(* CODESYS project OpenSML_TC3.library
   Company: Github
   DefaultNamespace: OpenSML
   Version: 3.2
   Placeholder: OpenSML
   Author: Feecat
   Description: Open Sources SoftMotion Light For CiA402 Servo Drivers
      visit https://github.com/feecat/OpenSML for more information
   Title: OpenSML

Project tree, tasks and I/O mapping:
  libraries: Tc2_Standard, * (Beckhoff Automation GmbH)
  S7RTT/
    function block FB_S7RTT_OTG [ST]
    function block FB_S7RTT_Plan [ST]
    function FC_S7RTT_AtTime [ST]
    function FC_S7RTT_BuildProfile [ST]
    function FC_S7RTT_CalcTrajDist [ST]
    data type ST_MotionLimits
    data type ST_MotionState
  data type OpenSML_Axis
  function block OpenSML_AxisController [ST]
  data type OpenSML_Control
  function block OpenSML_Home [ST]
  function block OpenSML_Power [ST]
  function block OpenSML_ProfilePosition [ST]
  function block OpenSML_ProfileVelocity [ST]
  function block OpenSML_Stop [ST]
  function block OpenSML_SyncPosition [ST]
  function block OpenSML_SyncVelocity [ST]
  function block OpenSML_TC3Link [ST]
*)

// S7RTT/ST_MotionLimits
TYPE ST_MotionLimits :
STRUCT
	fVelMax: LREAL;
	fAccMax: LREAL;
	fJerkMax: LREAL;
END_STRUCT
END_TYPE

// S7RTT/ST_MotionState
TYPE ST_MotionState :
STRUCT
	/// Duration of this segment 
	fDuration: LREAL := 0.0;
	/// Position 
	fPos: LREAL := 0.0;
	/// Velocity 
	fVel: LREAL := 0.0;
	/// Acceleration 
	fAcc: LREAL := 0.0;
	/// Jerk 
	fJerk: LREAL := 0.0;
END_STRUCT
END_TYPE

// OpenSML_Axis
TYPE OpenSML_Axis :
STRUCT
	///Output
	ControlWord: UINT;
	Modes_of_operation: SINT;
	Target_Position: DINT;
	Profile_Velocity: UDINT;
	Target_Velocity: DINT;
	Target_torque: INT;
	///Input
	StatusWord: UINT;
	Modes_of_operation_display: SINT;
	Torque_Actual_Value: INT;
	Position_Actual_Value: DINT;
	Velocity_Actual_Value: DINT;
	Current_Actual_Value: INT;
	Following_Error_Actual_Value: DINT;
END_STRUCT
END_TYPE

// OpenSML_Control
TYPE OpenSML_Control :
STRUCT
	///Axis Hardware Enable
	xAxisEnable: BOOL;
	///Jog&Pos Movement Enable
	xMoveEnable: BOOL;
	///Home Function Enable
	xHomeEnable: BOOL;
	///Simulation Mode
	xSimulation: BOOL;
	///Emergency Stop
	xEmergencyStop: BOOL := TRUE;
	///Jog Positive
	JogPos: BOOL;
	///Jog Negative
	JogNeg: BOOL;
	///Jog Velocity
	JogVelocity: LREAL := 10;
	///Actual Position Feedback
	lrActualPosition: LREAL;
	///Follow Target Position, Can be set to new value at any time
	lrFollowPosition: LREAL;
	///Follow Move Velocity, Can be set to new value at any time
	lrFollowVelocity: LREAL := 20;
	///Follow Move Enable
	xFollowEnable: BOOL;
	///Error
	xError: BOOL;
	///Busy, Normal Working State
	xBusy: BOOL;
	///In Position
	xInPosition: BOOL;
	///Axis Hardware Enabled
	xEnabled: BOOL;
	///Axis Home Done
	xHomeDone: BOOL;
	///Max Velocity
	MaxVelocity: LREAL := 100;
	///Max Acceleration
	MaxAcceleration: LREAL := 1000;
	///Max Jerk
	MaxJerk: LREAL := 10000;
	///Task Cycle Time, 0.001 = 1ms
	CycleTime: LREAL := 0.001;
	///Scale
	Scale: LREAL := 16#1000;
	///Axis Reference
	Axis: OpenSML_Axis;
END_STRUCT
END_TYPE

// S7RTT/FB_S7RTT_OTG
FUNCTION_BLOCK FB_S7RTT_OTG
VAR_INPUT
	///false=position, true=velocity
	ControlInterface: BOOL := FALSE;
	TargetPosition: LREAL;
	TargetVelocity: LREAL := 0;
	///1ms
	CycleTime: LREAL := 0.001;
	MaxVelocity: LREAL := 10;
	MaxAcceleration: LREAL := 10;
	MaxJerk: LREAL := 10;
	///set when init
	CurrentPosition: LREAL;
END_VAR
VAR_OUTPUT
	NewPosition: LREAL;
	NewVelocity: LREAL;
	NewAcceleration: LREAL;
	xError: BOOL;
END_VAR
VAR
	_ControlInterface: BOOL;
	_TargetPosition: LREAL;
	_TargetVelocity: LREAL;
	_CycleTime: LREAL;
	_MaxVelocity: LREAL;
	_MaxAcceleration: LREAL;
	_MaxJerk: LREAL;
	_CurrentPosition: LREAL;
	xExecute: BOOL;
	fbS7Planner: FB_S7RTT_Plan;
	stS7Limits: ST_MotionLimits;
	stS7Start: ST_MotionState;
	stS7Result: ST_MotionState;
	fS7Timer: LREAL;
END_VAR

// check if input changed
IF (ControlInterface <> _ControlInterface) OR
	(TargetPosition <> _TargetPosition) OR
	(TargetVelocity <> _TargetVelocity) OR
	(CycleTime <> _CycleTime) OR
	(MaxVelocity <> _MaxVelocity) OR
	(MaxAcceleration <> _MaxAcceleration) OR
	(MaxJerk <> _MaxJerk) OR
	(CurrentPosition <> _CurrentPosition) THEN
	
	IF CurrentPosition <> _CurrentPosition THEN
		stS7Start.fPos := CurrentPosition;
		stS7Result.fPos := CurrentPosition;
		_CurrentPosition := CurrentPosition;
	END_IF
	_ControlInterface := ControlInterface;
	_TargetPosition := TargetPosition;
	_TargetVelocity := TargetVelocity;
	_CycleTime := CycleTime;
	_MaxVelocity := MaxVelocity;
	_MaxAcceleration := MaxAcceleration;
	_MaxJerk := MaxJerk;
	
	xExecute:=TRUE;
END_IF

// main logic
IF xExecute THEN
    stS7Start.fPos := stS7Result.fPos;
    stS7Start.fVel := stS7Result.fVel;
    stS7Start.fAcc := stS7Result.fAcc;
    stS7Start.fDuration := 0.0;
    
    stS7Limits.fVelMax := MaxVelocity;
    stS7Limits.fAccMax := MaxAcceleration;
    stS7Limits.fJerkMax := MaxJerk;
    
    fbS7Planner.ModeVelocity := ControlInterface;
    fbS7Planner.StartState := stS7Start;
    fbS7Planner.TargetPos := TargetPosition;
    fbS7Planner.TargetVel := TargetVelocity; 
    fbS7Planner.Limits := stS7Limits;
    
    fS7Timer := 0.0;
END_IF

IF xExecute THEN
    fbS7Planner(Execute:=TRUE, Error=>xError);
    fbS7Planner(Execute:=FALSE);
END_IF

xExecute := FALSE;

fS7Timer := fS7Timer + CycleTime;

stS7Result := FC_S7RTT_AtTime(
	Trajectory := fbS7Planner.Trajectory, 
	SegCount := fbS7Planner.SegmentCount, 
	ElapsedTime := fS7Timer
);

NewPosition:=stS7Result.fPos;
NewVelocity:=stS7Result.fVel;
NewAcceleration:=stS7Result.fAcc;

END_FUNCTION_BLOCK

// S7RTT/FC_S7RTT_AtTime
FUNCTION FC_S7RTT_AtTime : ST_MotionState
VAR_INPUT
	Trajectory: ARRAY[1..32] OF ST_MotionState;
	SegCount: INT;
	ElapsedTime: LREAL;
END_VAR
VAR
	i: INT;
	t_rem: LREAL;
	t: LREAL;
	j: LREAL;
	p0: LREAL;
	v0: LREAL;
	a0: LREAL;
	last_idx: INT;
END_VAR

IF SegCount <= 0 THEN
    // No trajectory, return first state
    FC_S7RTT_AtTime.fPos := Trajectory[1].fPos; FC_S7RTT_AtTime.fVel := 0.0; FC_S7RTT_AtTime.fAcc := 0.0;
    RETURN;
END_IF;

IF ElapsedTime <= 0.0 THEN
     // Return Initial State from First Segment
     FC_S7RTT_AtTime := Trajectory[1]; 
     FC_S7RTT_AtTime.fDuration := 0.0;
     FC_S7RTT_AtTime.fJerk := 0.0;
     RETURN;
END_IF;

t_rem := ElapsedTime;

FOR i := 1 TO SegCount DO
	IF t_rem <= Trajectory[i].fDuration THEN
		t := t_rem;
		j := Trajectory[i].fJerk;
		// Use pre-calculated state at segment start
		p0 := Trajectory[i].fPos;
		v0 := Trajectory[i].fVel;
		a0 := Trajectory[i].fAcc;

		FC_S7RTT_AtTime.fPos := p0 + v0 * t + 0.5 * a0 * t*t + (1.0/6.0) * j * t*t*t;
		FC_S7RTT_AtTime.fVel := v0 + a0 * t + 0.5 * j * t*t;
		FC_S7RTT_AtTime.fAcc := a0 + j * t;
		FC_S7RTT_AtTime.fJerk := j;
		FC_S7RTT_AtTime.fDuration := 0.0;
		RETURN;
	ELSE
		t_rem := t_rem - Trajectory[i].fDuration;
	END_IF;
END_FOR;

// Time is beyond end of trajectory
// Calculate Final State of last segment
last_idx := SegCount;
t := Trajectory[last_idx].fDuration;
j := Trajectory[last_idx].fJerk;
p0 := Trajectory[last_idx].fPos;
v0 := Trajectory[last_idx].fVel;
a0 := Trajectory[last_idx].fAcc;

p0 := p0 + v0 * t + 0.5 * a0 * t*t + (1.0/6.0) * j * t*t*t;
v0 := v0 + a0 * t + 0.5 * j * t*t;

// Hold Final Position (assuming v=target, a=0 at end)
// Linear projection if Velocity is non-zero
FC_S7RTT_AtTime.fPos := p0 + v0 * t_rem;
FC_S7RTT_AtTime.fVel := v0;
FC_S7RTT_AtTime.fAcc := 0.0;
FC_S7RTT_AtTime.fJerk := 0.0;
FC_S7RTT_AtTime.fDuration := 0.0;

END_FUNCTION

// S7RTT/FB_S7RTT_Plan
FUNCTION_BLOCK FB_S7RTT_Plan
VAR_INPUT
	Execute: BOOL;
	ModeVelocity: BOOL;
	StartState: ST_MotionState;
	TargetPos: LREAL;
	TargetVel: LREAL;
	Limits: ST_MotionLimits;
END_VAR
VAR_OUTPUT
	Done: BOOL;
	Error: BOOL;
	SegmentCount: INT;
	Trajectory: ARRAY[1..32] OF ST_MotionState;
END_VAR
VAR
	/// State & Triggers
	trig_exec: BOOL;
	prev_exec: BOOL;
	c_pos: LREAL;
	c_vel: LREAL;
	c_acc: LREAL;
	/// Loop Iterators
	i: INT;
	/// Loop Iterators
	k: INT;
	/// General Calculation
	dist_req: LREAL;
	t_rec: LREAL;
	gap: LREAL;
	/// Check Bounds
	d_upper: LREAL;
	/// Check Bounds
	d_lower: LREAL;
	t_cruise: LREAL;
	/// --- Solver Shared Variables ---
	iter: INT;
	sa: LREAL;
	sb: LREAL;
	sc: LREAL;
	fa: LREAL;
	fb: LREAL;
	fc: LREAL;
	sd: LREAL;
	se: LREAL;
	tol1: LREAL;
	xm: LREAL;
	min1: LREAL;
	min2: LREAL;
	fCoefP: LREAL;
	fCoefQ: LREAL;
	fCoefR: LREAL;
	fCoefS: LREAL;
	mflag: BOOL;
	/// --- V1.7 Time Optimal Specific ---
	use_optimal: BOOL;
	opt_success: BOOL;
	/// 0 or 1
	j_idx: INT;
	j_apply: LREAL;
	search_horizon: LREAL;
	t_est: LREAL;
	/// Simulation / Cost Function Vars
	sim_p: LREAL;
	/// Simulation / Cost Function Vars
	sim_v: LREAL;
	/// Simulation / Cost Function Vars
	sim_a: LREAL;
	limit_a: LREAL;
	dist_to_lim: LREAL;
	t_ramp: LREAL;
	t_hold: LREAL;
	sat_dt: LREAL;
	sat_j: LREAL;
	/// Best Candidate Tracking
	valid_curr: BOOL;
	best_t_curr: LREAL;
	dur_curr: LREAL;
	winner_found: BOOL;
	winner_dur: LREAL;
	winner_t: LREAL;
	winner_j: LREAL;
	/// --- Fallback / Old Variables ---
	best_v: LREAL;
	v_mid: LREAL;
	a_mid: LREAL;
	v_inertial: LREAL;
	d_inertial: LREAL;
	t_to_zero: LREAL;
	j_restore: LREAL;
	/// Buffers
	t_shape_buf: ARRAY[1..5] OF LREAL;
	j_shape_buf: ARRAY[1..5] OF LREAL;
	shape_cnt: INT;
	/// Refinement
	ref_idx: INT;
	max_dt: LREAL;
	dt_fix: LREAL;
	v_cruise_start: LREAL;
	/// Constants (Updated V1.7)
	EPS_TIME: LREAL := 1E-10;
	/// Velocity Tolerance
	EPS_VAL: LREAL := 1E-10;
	EPS_ACC: LREAL := 1E-10;
	EPS_DIST: LREAL := 1E-10;
	MATH_EPS: LREAL := 1E-10;
	SOLVER_TOL: LREAL := 1E-10;
	SOLVER_EPS: LREAL := 2.22E-16;
	/// For initial checks
	SOLVER_COARSE: LREAL := 0.0001;
	MAX_ITER: INT := 50;
END_VAR

// ==============================================================================
// File Name:    FB_S7RTT_Plan.st
// Author:       feecat
// Version:      V1.8.1
// Description:  Simple 7seg Real-Time Trajectory Generator
// Website:      https://github.com/feecat/S7RTT
// License:      Apache License Version 2.0
// ==============================================================================
//
// Licensed under the Apache License, Version 2.0 (the "License");
// you may not use this file except in compliance with the License.
// You may obtain a copy of the License at
//
//     http://www.apache.org/licenses/LICENSE-2.0
//
// Unless required by applicable law or agreed to in writing, software
// distributed under the License is distributed on an "AS IS" BASIS,
// WITHOUT WARRANTIES OR CONDITIONS OF ANY KIND, either express or implied.
// See the License for the specific language governing permissions and
// limitations under the License.
// ==============================================================================

trig_exec := Execute AND NOT prev_exec;
prev_exec := Execute;

IF NOT Execute THEN
	Done := FALSE; Error := FALSE; RETURN;
END_IF

IF NOT trig_exec THEN RETURN; END_IF;

// --- Initialization ---
Done := FALSE;
Error := FALSE;
SegmentCount := 0;
opt_success := FALSE;

IF Limits.fVelMax <= 0.0 OR Limits.fAccMax <= 0.0 OR Limits.fJerkMax <= 0.0 THEN
	Error := TRUE; RETURN;
END_IF;

c_pos := StartState.fPos; c_vel := StartState.fVel; c_acc := StartState.fAcc;

// ========================================================
// 1. Acceleration Recovery (Safety Decel)
// ========================================================
IF c_acc > Limits.fAccMax + EPS_ACC THEN
	// Positive Saturation: Accel is too high positive, must reduce
	j_restore := -Limits.fJerkMax;
	limit_a := Limits.fAccMax;
	t_rec := (c_acc - limit_a) / (-j_restore);
	
	IF t_rec > EPS_TIME THEN
		SegmentCount := SegmentCount + 1;
		Trajectory[SegmentCount].fDuration := t_rec;
		Trajectory[SegmentCount].fJerk     := j_restore;
		// Integ State
		c_pos := c_pos + c_vel * t_rec + 0.5 * c_acc * t_rec*t_rec + (1.0/6.0) * j_restore * t_rec*t_rec*t_rec;
		c_vel := c_vel + c_acc * t_rec + 0.5 * j_restore * t_rec*t_rec;
		c_acc := limit_a;
	END_IF;
	
ELSIF c_acc < -Limits.fAccMax - EPS_ACC THEN
	// Negative Saturation: Accel is too low negative, must increase
	j_restore := Limits.fJerkMax;
	limit_a := -Limits.fAccMax;
	t_rec := (c_acc - limit_a) / (-j_restore); // Note: -j_restore here implies dividing by -JerkMax which is negative
	
	IF t_rec > EPS_TIME THEN
		SegmentCount := SegmentCount + 1;
		Trajectory[SegmentCount].fDuration := t_rec;
		Trajectory[SegmentCount].fJerk     := j_restore;
		// Integ State
		c_pos := c_pos + c_vel * t_rec + 0.5 * c_acc * t_rec*t_rec + (1.0/6.0) * j_restore * t_rec*t_rec*t_rec;
		c_vel := c_vel + c_acc * t_rec + 0.5 * j_restore * t_rec*t_rec;
		c_acc := limit_a;
	END_IF;
END_IF;

// ========================================================
// 2. Plan Generation
// ========================================================
IF ModeVelocity THEN
	// --- Velocity Mode (Unchanged Logic, New Constants) ---
	v_mid := TargetVel; 
	IF v_mid > Limits.fVelMax THEN v_mid := Limits.fVelMax; END_IF;
	IF v_mid < -Limits.fVelMax THEN v_mid := -Limits.fVelMax; END_IF;

	shape_cnt := FC_S7RTT_BuildProfile(c_vel, c_acc, v_mid, Limits.fAccMax, Limits.fJerkMax, t_shape_buf, j_shape_buf);
	IF shape_cnt > 0 THEN
		FOR i := 1 TO shape_cnt DO
			IF SegmentCount < 32 THEN
				SegmentCount := SegmentCount + 1;
				Trajectory[SegmentCount].fDuration := t_shape_buf[i];
				Trajectory[SegmentCount].fJerk     := j_shape_buf[i];
			END_IF;
		END_FOR;
	ELSE
		FOR i := 1 TO 31 DO
			SegmentCount := SegmentCount + 1;
			Trajectory[SegmentCount].fDuration := 0;
			Trajectory[SegmentCount].fJerk     := 0;
		END_FOR;
	END_IF
ELSE
	// --- Position Mode ---
	dist_req := TargetPos - c_pos;

	// Capacity Check (Can we reach target without hitting velocity limits?)
	// Note: FC_S7RTT_CalcTrajDist returns distance traveled to reach TargetVel via +/- VelMax
	d_upper := FC_S7RTT_CalcTrajDist(Limits.fVelMax, c_vel, c_acc, TargetVel, Limits.fAccMax, Limits.fJerkMax);
	d_lower := FC_S7RTT_CalcTrajDist(-Limits.fVelMax, c_vel, c_acc, TargetVel, Limits.fAccMax, Limits.fJerkMax);

	// Decision: Cruise or Optimal?
	use_optimal := TRUE;
	IF dist_req > d_upper + EPS_DIST THEN use_optimal := FALSE; END_IF;
	IF dist_req < d_lower - EPS_DIST THEN use_optimal := FALSE; END_IF;

	// ========================================================
	// 2.1 Time Optimal Solver (New V1.7 Feature)
	// ========================================================
	IF use_optimal THEN
		winner_found := FALSE;
		winner_dur := 1.0E10; // Init Large
		
		// Estimate search horizon
		t_est := (ABS(c_vel) + Limits.fVelMax) / Limits.fAccMax;
		IF t_est < 1.0 THEN t_est := 1.0; END_IF;
		search_horizon := t_est * 2.0 + 5.0;

		// Bidirectional Competition: Try +Jerk and -Jerk
		FOR j_idx := 0 TO 1 DO
			IF j_idx = 0 THEN j_apply := Limits.fJerkMax; ELSE j_apply := -Limits.fJerkMax; END_IF;
			valid_curr := FALSE;
			
			// Brent Solver Setup: Range [0, search_horizon]
			sa := 0.0; sb := search_horizon;
			
			// --- Evaluate at sa (0.0) ---
			// Inline Simulation Block 1
			sim_p := c_pos; sim_v := c_vel; sim_a := c_acc; // Reset State
			// Integrate Saturated (t=0 -> no effect), then Build Profile
			shape_cnt := FC_S7RTT_BuildProfile(sim_v, sim_a, TargetVel, Limits.fAccMax, Limits.fJerkMax, t_shape_buf, j_shape_buf);
			FOR k:=1 TO shape_cnt DO 
				sim_p := sim_p + sim_v*t_shape_buf[k] + 0.5*sim_a*t_shape_buf[k]*t_shape_buf[k] + (1.0/6.0)*j_shape_buf[k]*t_shape_buf[k]*t_shape_buf[k]*t_shape_buf[k]; 
				sim_v := sim_v + sim_a*t_shape_buf[k] + 0.5*j_shape_buf[k]*t_shape_buf[k]*t_shape_buf[k];
				sim_a := sim_a + j_shape_buf[k]*t_shape_buf[k];
			END_FOR;
			fa := sim_p - TargetPos; // Error at t=0
			
			IF ABS(fa) < SOLVER_COARSE THEN
				best_t_curr := 0.0; valid_curr := TRUE;
			ELSE
				// --- Evaluate at sb (horizon) ---
				// Inline Simulation Block 2
				sim_p := c_pos; sim_v := c_vel; sim_a := c_acc;
				limit_a := Limits.fAccMax; IF j_apply < 0 THEN limit_a := -Limits.fAccMax; END_IF;
				dist_to_lim := limit_a - sim_a;
				IF (j_apply > 0 AND dist_to_lim > -MATH_EPS) OR (j_apply < 0 AND dist_to_lim < MATH_EPS) THEN t_ramp := dist_to_lim / j_apply; ELSE t_ramp := 0.0; END_IF;
				// Saturated Int (simplified logic for end of range)
				IF sb <= t_ramp THEN
					sim_p:=sim_p+sim_v*sb+0.5*sim_a*sb*sb+(1.0/6.0)*j_apply*sb*sb*sb; sim_v:=sim_v+sim_a*sb+0.5*j_apply*sb*sb; sim_a:=sim_a+j_apply*sb;
				ELSE
					sim_p:=sim_p+sim_v*t_ramp+0.5*sim_a*t_ramp*t_ramp+(1.0/6.0)*j_apply*t_ramp*t_ramp*t_ramp; sim_v:=sim_v+sim_a*t_ramp+0.5*j_apply*t_ramp*t_ramp; sim_a:=sim_a+j_apply*t_ramp;
					sim_a:=limit_a; t_hold:=sb-t_ramp;
					sim_p:=sim_p+sim_v*t_hold+0.5*sim_a*t_hold*t_hold; sim_v:=sim_v+sim_a*t_hold;
				END_IF;
				shape_cnt := FC_S7RTT_BuildProfile(sim_v, sim_a, TargetVel, Limits.fAccMax, Limits.fJerkMax, t_shape_buf, j_shape_buf);
				FOR k:=1 TO shape_cnt DO sim_p:=sim_p+sim_v*t_shape_buf[k]+0.5*sim_a*t_shape_buf[k]*t_shape_buf[k]+(1.0/6.0)*j_shape_buf[k]*t_shape_buf[k]*t_shape_buf[k]*t_shape_buf[k]; sim_v:=sim_v+sim_a*t_shape_buf[k]+0.5*j_shape_buf[k]*t_shape_buf[k]*t_shape_buf[k]; sim_a:=sim_a+j_shape_buf[k]*t_shape_buf[k]; END_FOR;
				fb := sim_p - TargetPos;

				// Bounds Check
				IF fa * fb <= 0.0 THEN
					// Brent Loop
					sc := sa; fc := fa; sd := sb - sa; se := sd; mflag := TRUE;
					FOR iter := 1 TO MAX_ITER DO
						IF ABS(fc) < ABS(fb) THEN sa:=sb; sb:=sc; sc:=sa; fa:=fb; fb:=fc; fc:=fa; END_IF;
						tol1 := 2.0 * SOLVER_EPS * ABS(sb) + 0.5 * SOLVER_TOL; xm := 0.5 * (sc - sb);
						IF ABS(xm) <= tol1 OR fb = 0.0 THEN EXIT; END_IF;
						IF ABS(se) >= tol1 AND ABS(fa) > ABS(fb) THEN
							fCoefS := fb / fa;
							IF sa = sc THEN fCoefP := 2.0*xm*fCoefS; fCoefQ := 1.0-fCoefS;
							ELSE fCoefQ := fa/fc; fCoefR := fb/fc; fCoefP := fCoefS*(2.0*xm*fCoefQ*(fCoefQ-fCoefR)-(sb-sa)*(fCoefR-1.0)); fCoefQ := (fCoefQ-1.0)*(fCoefR-1.0)*(fCoefS-1.0); END_IF;
							IF fCoefP > 0.0 THEN fCoefQ := -fCoefQ; END_IF; fCoefP := ABS(fCoefP);
							min1 := 3.0*xm*fCoefQ - ABS(tol1*fCoefQ); min2 := ABS(se*fCoefQ);
							IF 2.0*fCoefP < min1 THEN
								IF mflag THEN IF 2.0*fCoefP < min2 THEN se:=sd; sd:=fCoefP/fCoefQ; mflag:=FALSE; ELSE sd:=xm; se:=sd; mflag:=TRUE; END_IF;
								ELSE IF 2.0*fCoefP < ABS(sd*fCoefQ) THEN se:=sd; sd:=fCoefP/fCoefQ; mflag:=FALSE; ELSE sd:=xm; se:=sd; mflag:=TRUE; END_IF; END_IF;
							ELSE sd:=xm; se:=sd; mflag:=TRUE; END_IF;
						ELSE sd:=xm; se:=sd; mflag:=TRUE; END_IF;
						sa := sb; fa := fb;
						IF ABS(sd) > tol1 THEN sb:=sb+sd; ELSE IF xm > 0.0 THEN sb:=sb+tol1; ELSE sb:=sb-tol1; END_IF; END_IF;
						
						// --- Eval Function (t = sb) ---
						// Only necessary to update fb. Re-use simulation logic.
						sim_p := c_pos; sim_v := c_vel; sim_a := c_acc;
						limit_a := Limits.fAccMax; IF j_apply < 0 THEN limit_a := -Limits.fAccMax; END_IF;
						dist_to_lim := limit_a - sim_a;
						IF (j_apply > 0 AND dist_to_lim > -MATH_EPS) OR (j_apply < 0 AND dist_to_lim < MATH_EPS) THEN t_ramp := dist_to_lim / j_apply; ELSE t_ramp := 0.0; END_IF;
						IF sb <= t_ramp THEN
							IF sb > EPS_TIME THEN sim_p:=sim_p+sim_v*sb+0.5*sim_a*sb*sb+(1.0/6.0)*j_apply*sb*sb*sb; sim_v:=sim_v+sim_a*sb+0.5*j_apply*sb*sb; sim_a:=sim_a+j_apply*sb; END_IF;
						ELSE
							IF t_ramp > EPS_TIME THEN sim_p:=sim_p+sim_v*t_ramp+0.5*sim_a*t_ramp*t_ramp+(1.0/6.0)*j_apply*t_ramp*t_ramp*t_ramp; sim_v:=sim_v+sim_a*t_ramp+0.5*j_apply*t_ramp*t_ramp; sim_a:=sim_a+j_apply*t_ramp; END_IF;
							sim_a:=limit_a; t_hold:=sb-t_ramp;
							IF t_hold > EPS_TIME THEN sim_p:=sim_p+sim_v*t_hold+0.5*sim_a*t_hold*t_hold; sim_v:=sim_v+sim_a*t_hold; END_IF;
						END_IF;
						shape_cnt := FC_S7RTT_BuildProfile(sim_v, sim_a, TargetVel, Limits.fAccMax, Limits.fJerkMax, t_shape_buf, j_shape_buf);
						FOR k:=1 TO shape_cnt DO sim_p:=sim_p+sim_v*t_shape_buf[k]+0.5*sim_a*t_shape_buf[k]*t_shape_buf[k]+(1.0/6.0)*j_shape_buf[k]*t_shape_buf[k]*t_shape_buf[k]*t_shape_buf[k]; sim_v:=sim_v+sim_a*t_shape_buf[k]+0.5*j_shape_buf[k]*t_shape_buf[k]*t_shape_buf[k]; sim_a:=sim_a+j_shape_buf[k]*t_shape_buf[k]; END_FOR;
						fb := sim_p - TargetPos;
						// --- End Eval ---
						
						IF (fb > 0.0 AND fc > 0.0) OR (fb < 0.0 AND fc < 0.0) THEN sc := sa; fc := fa; sd := sb - sa; se := sd; mflag := TRUE; END_IF;
					END_FOR;
					best_t_curr := sb;
					IF ABS(fb) <= SOLVER_COARSE THEN valid_curr := TRUE; END_IF;
				END_IF;
			END_IF;
			
			// Calculate Total Duration for Comparison
			IF valid_curr THEN
				dur_curr := 0.0;
				// Saturated Time
				limit_a := Limits.fAccMax; IF j_apply < 0 THEN limit_a := -Limits.fAccMax; END_IF;
				dist_to_lim := limit_a - c_acc;
				IF (j_apply > 0 AND dist_to_lim > -MATH_EPS) OR (j_apply < 0 AND dist_to_lim < MATH_EPS) THEN t_ramp := dist_to_lim / j_apply; ELSE t_ramp := 0.0; END_IF;
				IF best_t_curr <= t_ramp THEN dur_curr := best_t_curr;
				ELSE dur_curr := best_t_curr; // t_ramp + (t - t_ramp)
				END_IF;
				// Sim to get intermediate state for remaining profile
				sim_p := c_pos; sim_v := c_vel; sim_a := c_acc;
				IF best_t_curr <= t_ramp THEN
					IF best_t_curr > EPS_TIME THEN sim_v:=sim_v+sim_a*best_t_curr+0.5*j_apply*best_t_curr*best_t_curr; sim_a:=sim_a+j_apply*best_t_curr; END_IF;
				ELSE
					IF t_ramp > EPS_TIME THEN sim_v:=sim_v+sim_a*t_ramp+0.5*j_apply*t_ramp*t_ramp; sim_a:=sim_a+j_apply*t_ramp; END_IF;
					sim_a:=limit_a; t_hold:=best_t_curr-t_ramp;
					IF t_hold > EPS_TIME THEN sim_v:=sim_v+sim_a*t_hold; END_IF;
				END_IF;
				shape_cnt := FC_S7RTT_BuildProfile(sim_v, sim_a, TargetVel, Limits.fAccMax, Limits.fJerkMax, t_shape_buf, j_shape_buf);
				FOR k:=1 TO shape_cnt DO dur_curr := dur_curr + t_shape_buf[k]; END_FOR;
				
				// Update Winner
				IF dur_curr < winner_dur THEN winner_dur := dur_curr; winner_t := best_t_curr; winner_j := j_apply; winner_found := TRUE; END_IF;
			END_IF;
		END_FOR;
		
		// Construct Winner
		IF winner_found THEN
			opt_success := TRUE;
			limit_a := Limits.fAccMax; IF winner_j < 0 THEN limit_a := -Limits.fAccMax; END_IF;
			dist_to_lim := limit_a - c_acc;
			IF (winner_j > 0 AND dist_to_lim > -MATH_EPS) OR (winner_j < 0 AND dist_to_lim < MATH_EPS) THEN t_ramp := dist_to_lim / winner_j; ELSE t_ramp := 0.0; END_IF;
			
			IF winner_t <= t_ramp THEN
				IF winner_t > EPS_TIME THEN
					IF SegmentCount < 32 THEN SegmentCount:=SegmentCount+1; Trajectory[SegmentCount].fDuration:=winner_t; Trajectory[SegmentCount].fJerk:=winner_j; END_IF;
					c_pos:=c_pos+c_vel*winner_t+0.5*c_acc*winner_t*winner_t+(1.0/6.0)*winner_j*winner_t*winner_t*winner_t; c_vel:=c_vel+c_acc*winner_t+0.5*winner_j*winner_t*winner_t; c_acc:=c_acc+winner_j*winner_t;
				END_IF;
			ELSE
				IF t_ramp > EPS_TIME THEN
					IF SegmentCount < 32 THEN SegmentCount:=SegmentCount+1; Trajectory[SegmentCount].fDuration:=t_ramp; Trajectory[SegmentCount].fJerk:=winner_j; END_IF;
					c_pos:=c_pos+c_vel*t_ramp+0.5*c_acc*t_ramp*t_ramp+(1.0/6.0)*winner_j*t_ramp*t_ramp*t_ramp; c_vel:=c_vel+c_acc*t_ramp+0.5*winner_j*t_ramp*t_ramp; c_acc:=c_acc+winner_j*t_ramp;
				END_IF;
				c_acc := limit_a; t_hold := winner_t - t_ramp;
				IF t_hold > EPS_TIME THEN
					IF SegmentCount < 32 THEN SegmentCount:=SegmentCount+1; Trajectory[SegmentCount].fDuration:=t_hold; Trajectory[SegmentCount].fJerk:=0.0; END_IF;
					c_pos:=c_pos+c_vel*t_hold+0.5*c_acc*t_hold*t_hold; c_vel:=c_vel+c_acc*t_hold;
				END_IF;
			END_IF;
			shape_cnt := FC_S7RTT_BuildProfile(c_vel, c_acc, TargetVel, Limits.fAccMax, Limits.fJerkMax, t_shape_buf, j_shape_buf);
			FOR i:=1 TO shape_cnt DO IF SegmentCount < 32 THEN SegmentCount:=SegmentCount+1; Trajectory[SegmentCount].fDuration:=t_shape_buf[i]; Trajectory[SegmentCount].fJerk:=j_shape_buf[i]; END_IF; END_FOR;
		END_IF;
	END_IF;

	// ========================================================
	// 2.2 Fallback / Cruise Logic (Original + Cruise)
	// ========================================================
	IF NOT opt_success THEN
		// If dist_req > d_upper, we Cruise at VMax. If < d_lower, at -VMax. 
		// Otherwise, we solve for intermediate peak.
		
		IF dist_req > d_upper + EPS_DIST THEN best_v := Limits.fVelMax;
		ELSIF dist_req < d_lower - EPS_DIST THEN best_v := -Limits.fVelMax;
		ELSE
			// Bisection Solver (Original Logic, compacted)
			sa := -Limits.fVelMax; sb := Limits.fVelMax;
			// Calc Fa/Fb using helper function logic (Dist via profile)
			// Note: Assuming FC_S7RTT_CalcTrajDist calculates distance for a profile peaking at 'sa'/'sb' then going to TargetVel
			fa := FC_S7RTT_CalcTrajDist(sa, c_vel, c_acc, TargetVel, Limits.fAccMax, Limits.fJerkMax) - dist_req;
			fb := FC_S7RTT_CalcTrajDist(sb, c_vel, c_acc, TargetVel, Limits.fAccMax, Limits.fJerkMax) - dist_req;
			
			IF fa * fb > 0.0 THEN IF ABS(fa) < ABS(fb) THEN best_v := sa; ELSE best_v := sb; END_IF;
			ELSE
				sc:=sa; fc:=fa; sd:=sb-sa; se:=sd; mflag:=TRUE;
				FOR iter := 1 TO MAX_ITER DO
					IF ABS(fc) < ABS(fb) THEN sa:=sb; sb:=sc; sc:=sa; fa:=fb; fb:=fc; fc:=fa; END_IF;
					tol1 := 2.0 * SOLVER_EPS * ABS(sb) + 0.5 * SOLVER_TOL; xm := 0.5 * (sc - sb);
					IF ABS(xm) <= tol1 OR fb = 0.0 THEN EXIT; END_IF;
					IF ABS(se) >= tol1 AND ABS(fa) > ABS(fb) THEN
						fCoefS := fb/fa;
						IF sa=sc THEN fCoefP:=2.0*xm*fCoefS; fCoefQ:=1.0-fCoefS; ELSE fCoefQ:=fa/fc; fCoefR:=fb/fc; fCoefP:=fCoefS*(2.0*xm*fCoefQ*(fCoefQ-fCoefR)-(sb-sa)*(fCoefR-1.0)); fCoefQ:=(fCoefQ-1.0)*(fCoefR-1.0)*(fCoefS-1.0); END_IF;
						IF fCoefP > 0.0 THEN fCoefQ:=-fCoefQ; END_IF; fCoefP:=ABS(fCoefP); min1:=3.0*xm*fCoefQ-ABS(tol1*fCoefQ); min2:=ABS(se*fCoefQ);
						IF 2.0*fCoefP < min1 THEN IF mflag THEN IF 2.0*fCoefP < min2 THEN se:=sd; sd:=fCoefP/fCoefQ; mflag:=FALSE; ELSE sd:=xm; se:=sd; mflag:=TRUE; END_IF; ELSE IF 2.0*fCoefP < ABS(sd*fCoefQ) THEN se:=sd; sd:=fCoefP/fCoefQ; mflag:=FALSE; ELSE sd:=xm; se:=sd; mflag:=TRUE; END_IF; END_IF; ELSE sd:=xm; se:=sd; mflag:=TRUE; END_IF;
					ELSE sd:=xm; se:=sd; mflag:=TRUE; END_IF;
					sa:=sb; fa:=fb; IF ABS(sd) > tol1 THEN sb:=sb+sd; ELSE IF xm > 0.0 THEN sb:=sb+tol1; ELSE sb:=sb-tol1; END_IF; END_IF;
					fb := FC_S7RTT_CalcTrajDist(sb, c_vel, c_acc, TargetVel, Limits.fAccMax, Limits.fJerkMax) - dist_req;
					IF (fb > 0.0 AND fc > 0.0) OR (fb < 0.0 AND fc < 0.0) THEN sc:=sa; fc:=fa; sd:=sb-sa; se:=sd; mflag:=TRUE; END_IF;
				END_FOR;
				best_v := sb;
			END_IF;
		END_IF;

		// Generate fallback profile
		shape_cnt := FC_S7RTT_BuildProfile(c_vel, c_acc, best_v, Limits.fAccMax, Limits.fJerkMax, t_shape_buf, j_shape_buf);
		FOR i:=1 TO shape_cnt DO
			IF SegmentCount < 32 THEN SegmentCount:=SegmentCount+1; Trajectory[SegmentCount].fDuration:=t_shape_buf[i]; Trajectory[SegmentCount].fJerk:=j_shape_buf[i]; END_IF;
			c_pos:=c_pos+c_vel*t_shape_buf[i]+0.5*c_acc*t_shape_buf[i]*t_shape_buf[i]+(1.0/6.0)*j_shape_buf[i]*t_shape_buf[i]*t_shape_buf[i]*t_shape_buf[i];
			c_vel:=c_vel+c_acc*t_shape_buf[i]+0.5*j_shape_buf[i]*t_shape_buf[i]*t_shape_buf[i]; c_acc:=c_acc+j_shape_buf[i]*t_shape_buf[i];
		END_FOR;
		// Add Cruise if needed (gap logic)
		c_acc := 0.0; 
		// Sim fwd
		sim_p := c_pos; sim_v := c_vel; sim_a := 0.0;
		shape_cnt := FC_S7RTT_BuildProfile(sim_v, sim_a, TargetVel, Limits.fAccMax, Limits.fJerkMax, t_shape_buf, j_shape_buf);
		FOR k:=1 TO shape_cnt DO sim_p:=sim_p+sim_v*t_shape_buf[k]+0.5*sim_a*t_shape_buf[k]*t_shape_buf[k]+(1.0/6.0)*j_shape_buf[k]*t_shape_buf[k]*t_shape_buf[k]*t_shape_buf[k]; sim_v:=sim_v+sim_a*t_shape_buf[k]+0.5*j_shape_buf[k]*t_shape_buf[k]*t_shape_buf[k]; sim_a:=sim_a+j_shape_buf[k]*t_shape_buf[k]; END_FOR;
		gap := TargetPos - sim_p;
		IF ABS(c_vel) > EPS_VAL AND ABS(gap) > EPS_DIST THEN
			t_cruise := gap / c_vel;
			IF t_cruise > EPS_TIME THEN
				IF SegmentCount < 32 THEN SegmentCount:=SegmentCount+1; Trajectory[SegmentCount].fDuration:=t_cruise; Trajectory[SegmentCount].fJerk:=0.0; END_IF;
				c_pos := c_pos + c_vel * t_cruise;
			END_IF;
		END_IF;
		// Final Decel
		shape_cnt := FC_S7RTT_BuildProfile(c_vel, c_acc, TargetVel, Limits.fAccMax, Limits.fJerkMax, t_shape_buf, j_shape_buf);
		FOR i:=1 TO shape_cnt DO IF SegmentCount < 32 THEN SegmentCount:=SegmentCount+1; Trajectory[SegmentCount].fDuration:=t_shape_buf[i]; Trajectory[SegmentCount].fJerk:=j_shape_buf[i]; END_IF; END_FOR;
	END_IF;
END_IF;

// ========================================================
// 2.5 Trajectory Refinement (Precision Fix)
// ========================================================
IF SegmentCount > 0 AND NOT ModeVelocity THEN
	c_pos := StartState.fPos; c_vel := StartState.fVel; c_acc := StartState.fAcc;
	ref_idx := -1; max_dt := -1.0;
	FOR i := 1 TO SegmentCount DO
		t_rec := Trajectory[i].fDuration; j_restore := Trajectory[i].fJerk;
		IF ABS(j_restore) < MATH_EPS AND ABS(c_acc) < EPS_ACC THEN IF t_rec > max_dt THEN max_dt:=t_rec; ref_idx:=i; v_cruise_start:=c_vel; END_IF; END_IF;
		c_pos:=c_pos+c_vel*t_rec+0.5*c_acc*t_rec*t_rec+(1.0/6.0)*j_restore*t_rec*t_rec*t_rec; c_vel:=c_vel+c_acc*t_rec+0.5*j_restore*t_rec*t_rec; c_acc:=c_acc+j_restore*t_rec;
	END_FOR;
	gap := TargetPos - c_pos;
	IF ref_idx <> -1 AND ABS(gap) > EPS_DIST AND ABS(v_cruise_start) > EPS_VAL THEN
		dt_fix := gap / v_cruise_start;
		Trajectory[ref_idx].fDuration := Trajectory[ref_idx].fDuration + dt_fix;
		IF Trajectory[ref_idx].fDuration < EPS_TIME THEN Trajectory[ref_idx].fDuration := EPS_TIME; END_IF;
	END_IF;
END_IF;

// ========================================================
// 3. Final Pass
// ========================================================
c_pos := StartState.fPos; c_vel := StartState.fVel; c_acc := StartState.fAcc;
FOR i := 1 TO SegmentCount DO
	Trajectory[i].fPos := c_pos; Trajectory[i].fVel := c_vel; Trajectory[i].fAcc := c_acc;
	t_rec := Trajectory[i].fDuration; j_restore := Trajectory[i].fJerk;
	c_pos:=c_pos+c_vel*t_rec+0.5*c_acc*t_rec*t_rec+(1.0/6.0)*j_restore*t_rec*t_rec*t_rec; c_vel:=c_vel+c_acc*t_rec+0.5*j_restore*t_rec*t_rec; c_acc:=c_acc+j_restore*t_rec;
END_FOR;

IF SegmentCount = 0 THEN
	Trajectory[1]:= StartState;
	Trajectory[1].fDuration := 0; Trajectory[1].fJerk := 0; Trajectory[1].fAcc := 0;
	SegmentCount := 1;
END_IF

Done := TRUE;
Done := TRUE;

END_FUNCTION_BLOCK

// S7RTT/FC_S7RTT_BuildProfile
FUNCTION FC_S7RTT_BuildProfile : INT
VAR_INPUT
	in_v_start: LREAL;
	in_a_start: LREAL;
	in_v_target: LREAL;
	in_a_max: LREAL;
	in_j_max: LREAL;
END_VAR
VAR_IN_OUT
	out_time: ARRAY[1..5] OF LREAL;
	out_jerk: ARRAY[1..5] OF LREAL;
END_VAR
VAR
	acc_clamped: LREAL;
	t_to_zero: LREAL;
	j_restore: LREAL;
	v_min_feasible: LREAL;
	direction: LREAL;
	v0_mod: LREAL;
	a0_mod: LREAL;
	v1_mod: LREAL;
	t1_max: LREAL;
	t3_max: LREAL;
	dv_inflection: LREAL;
	dv_req: LREAL;
	dv_missing: LREAL;
	term: LREAL;
	a_peak: LREAL;
	t1: LREAL;
	t2: LREAL;
	t3: LREAL;
	cnt: INT;
	EPS: LREAL := 1E-10;
END_VAR

cnt := 0;

// 1. Clamp initial acceleration to limits
acc_clamped := in_a_start;
IF acc_clamped > in_a_max THEN acc_clamped := in_a_max; END_IF;
IF acc_clamped < -in_a_max THEN acc_clamped := -in_a_max; END_IF;

// 2. Check feasibility (can we stop?)
t_to_zero := ABS(acc_clamped) / in_j_max;
IF ABS(acc_clamped) > EPS THEN
    IF acc_clamped > 0.0 THEN j_restore := -in_j_max; ELSE j_restore := in_j_max; END_IF;
ELSE
    j_restore := 0.0;
END_IF;

v_min_feasible := in_v_start + acc_clamped * t_to_zero + 0.5 * j_restore * t_to_zero * t_to_zero;

// 3. Determine direction
direction := 1.0;
IF in_v_target < v_min_feasible - EPS THEN
    direction := -1.0;
END_IF;

// 4. Normalize to positive quadrant
v0_mod := in_v_start * direction;
a0_mod := acc_clamped * direction;
v1_mod := in_v_target * direction;

t1_max := (in_a_max - a0_mod) / in_j_max;
IF t1_max < 0.0 THEN t1_max := 0.0; END_IF;

t3_max := in_a_max / in_j_max;

// Velocity change at inflection (max accel reached)
dv_inflection := (a0_mod * t1_max + 0.5 * in_j_max * t1_max * t1_max) +
                 (in_a_max * t3_max - 0.5 * in_j_max * t3_max * t3_max);

dv_req := v1_mod - v0_mod;

// 5. Calculate profile times
IF dv_req > dv_inflection THEN
    // Trapezoidal (Constant Acceleration Phase)
    dv_missing := dv_req - dv_inflection;
    t2 := dv_missing / in_a_max;
    t1 := t1_max;
    t3 := t3_max;
ELSE
    // Triangular (No Constant Acceleration)
    term := in_j_max * dv_req + 0.5 * a0_mod * a0_mod;
    IF term < 0.0 THEN term := 0.0; END_IF;
    a_peak := SQRT(term);
    
    t1 := (a_peak - a0_mod) / in_j_max;
    IF t1 < 0.0 THEN t1 := 0.0; END_IF;
    
    t3 := a_peak / in_j_max;
    IF t3 < 0.0 THEN t3 := 0.0; END_IF;
    
    t2 := 0.0;
END_IF;

// 6. Output Segments
IF t1 > EPS THEN
    cnt := cnt + 1; out_time[cnt] := t1; out_jerk[cnt] := direction * in_j_max;
END_IF;
IF t2 > EPS THEN
    cnt := cnt + 1; out_time[cnt] := t2; out_jerk[cnt] := 0.0;
END_IF;
IF t3 > EPS THEN
    cnt := cnt + 1; out_time[cnt] := t3; out_jerk[cnt] := -direction * in_j_max;
END_IF;

FC_S7RTT_BuildProfile := cnt;

END_FUNCTION

// S7RTT/FC_S7RTT_CalcTrajDist
FUNCTION FC_S7RTT_CalcTrajDist : LREAL
VAR_INPUT
	v_peak: LREAL;
	start_v: LREAL;
	start_a: LREAL;
	target_v: LREAL;
	a_max: LREAL;
	j_max: LREAL;
END_VAR
VAR
	t_buf: ARRAY[1..5] OF LREAL;
	j_buf: ARRAY[1..5] OF LREAL;
	cnt: INT;
	i: INT;
	v_curr: LREAL;
	a_curr: LREAL;
	dist_total: LREAL;
	t_seg: LREAL;
	j_seg: LREAL;
END_VAR

dist_total := 0.0;
v_curr := start_v;
a_curr := start_a;

// Phase 1: Start -> Peak Velocity
cnt := FC_S7RTT_BuildProfile(v_curr, a_curr, v_peak, a_max, j_max, t_buf, j_buf);
FOR i := 1 TO cnt DO
	t_seg := t_buf[i];
	j_seg := j_buf[i];
    // Standard kinematic integration: p = p0 + v0*t + 0.5*a0*t^2 + 1/6*j*t^3
	dist_total := dist_total + v_curr * t_seg + 0.5 * a_curr * t_seg*t_seg + (1.0/6.0) * j_seg * t_seg*t_seg*t_seg;
	v_curr := v_curr + a_curr * t_seg + 0.5 * j_seg * t_seg*t_seg;
	a_curr := a_curr + j_seg * t_seg;
END_FOR;

// Phase 2: Peak Velocity -> Target Velocity
cnt := FC_S7RTT_BuildProfile(v_curr, a_curr, target_v, a_max, j_max, t_buf, j_buf);
FOR i := 1 TO cnt DO
	t_seg := t_buf[i];
	j_seg := j_buf[i];
	dist_total := dist_total + v_curr * t_seg + 0.5 * a_curr * t_seg*t_seg + (1.0/6.0) * j_seg * t_seg*t_seg*t_seg;
	v_curr := v_curr + a_curr * t_seg + 0.5 * j_seg * t_seg*t_seg;
	a_curr := a_curr + j_seg * t_seg;
END_FOR;

FC_S7RTT_CalcTrajDist := dist_total;

END_FUNCTION

// OpenSML_AxisController
/// https://github.com/feecat/opensml 
FUNCTION_BLOCK OpenSML_AxisController
VAR_IN_OUT
	Axis: OpenSML_Axis;
	Control: OpenSML_Control;
END_VAR
VAR
	Power: OpenSML_Power;
	Home: OpenSML_Home;
	iState: INT;
	otg: FB_S7RTT_OTG;
	InterfaceType: BOOL;
	JogVel: LREAL;
	MoveVel: LREAL;
END_VAR


Power(
	Axis:=Axis , 
	xEnable:=Control.xAxisEnable , 
	xEmergencyStop:=Control.xEmergencyStop , 
	xDone=>Control.xEnabled , 
	xError=> );

Home(
	Axis:=Axis , 
	xEnable:=Control.xHomeEnable AND NOT Control.xMoveEnable , 
	xDone=>Control.xHomeDone , 
	xError=> );

(*
Cyclic Synchronous Position Mode (=8)
Set 6060(Op mode) and 60C2(Interpolation time period) at Startup Parameters.

#####################################
NEED StruckigLight Library for Quadratic Velocity Ramp Calculate.

If in movement, Please DO NOT Drop down xEnable.
#####################################
*)

Control.xInPosition:=FALSE;

IF control.xSimulation THEN
	Axis.Position_Actual_Value:=Axis.Target_Position;
END_IF

control.lrActualPosition:=DINT_TO_LREAL(Axis.Position_Actual_Value) / Control.Scale;

CASE iState OF
	0://start
		Control.xError:=FALSE;
		IF Control.xMoveEnable AND Axis.StatusWord.1 AND Axis.StatusWord.2 AND Axis.Modes_of_operation_display = 8 AND NOT Axis.StatusWord.3 THEN//ready
			iState:=10;//go go
		ELSIF Control.xMoveEnable AND Axis.StatusWord.1 AND Axis.Modes_of_operation_display <> 8 THEN//need switch mode
			Axis.ControlWord.3:=FALSE;//drop down operation enabled, motor could free move
			iState:=10;
		ELSIF Control.xMoveEnable AND Control.xSimulation THEN
			iState:=20;
		ELSIF Control.xMoveEnable THEN
			iState:=999;//error
		END_IF
	10://Set Mode
		Axis.Modes_of_operation:=8;//Cyclic Synchronous Position Mode
		Axis.ControlWord.3:=Axis.Modes_of_operation_display=8;//Success change mode, enable operation
		otg.CurrentPosition:=DINT_TO_LREAL(Axis.Position_Actual_Value) / Control.Scale;//Write actual position to otg
		IF Axis.StatusWord.2 AND Axis.Modes_of_operation_display = 8 THEN//Operation Enabled, Mode Changed success
			iState:=20;
		END_IF
	20://Movement
		IF Control.JogPos AND NOT Control.xFollowEnable THEN
			InterfaceType:=1;
			JogVel:=MIN(Control.JogVelocity, Control.MaxVelocity);
		ELSIF Control.JogNeg AND NOT Control.xFollowEnable THEN
			InterfaceType:=1;
			JogVel:=MAX(-Control.JogVelocity, -Control.MaxVelocity);
		ELSE
			InterfaceType:=1;
			JogVel:=0;
		END_IF
		
		IF Control.xFollowEnable AND Control.lrFollowVelocity > 0 THEN
			InterfaceType:=0;
			MoveVel:=MIN(Control.lrFollowVelocity, Control.MaxVelocity);
		ELSE
			MoveVel:= Control.MaxVelocity;
		END_IF
		
		otg(
			ControlInterface:= InterfaceType,
			TargetPosition:= Control.lrFollowPosition , 
			TargetVelocity:= JogVel , 
			CycleTIme:= Control.CycleTime,
			MaxVelocity:= MoveVel,//Control.para.MaxVelocity , 
			MaxAcceleration:= Control.MaxAcceleration , 
			MaxJerk:= Control.MaxJerk);//accept new position and going on
			
		IF otg.NewPosition >= 0 THEN
			Axis.Target_Position := LREAL_TO_DINT(otg.NewPosition * Control.Scale);
		ELSE
			Axis.Target_Position := - LREAL_TO_DINT( - otg.NewPosition * Control.Scale);//it fix negative overflow problem.
		END_IF
		
		Control.xInPosition := ABS(otg.NewPosition - Control.lrActualPosition) < 0.01;
		
		IF Axis.StatusWord.13 OR Axis.StatusWord.3 OR otg.xError OR Power.xError OR Home.xError THEN//Axis Error
			iState:=999;
		ELSIF NOT Control.xMoveEnable THEN
			iState:=0;
		END_IF
	999://Error wait
		Control.xError:=TRUE;
		IF NOT Control.xMoveEnable THEN
			iState:=0;
		END_IF
END_CASE

END_FUNCTION_BLOCK

// OpenSML_Power
/// https://github.com/feecat/opensml 
FUNCTION_BLOCK OpenSML_Power
VAR_IN_OUT
	Axis: OpenSML_Axis;
END_VAR
VAR_INPUT
	xEnable: BOOL;
	xEmergencyStop: BOOL := TRUE;
END_VAR
VAR_OUTPUT
	xDone: BOOL;
	xError: BOOL;
END_VAR
VAR
	iState: INT;
	tonTimeout: TON;
	tTimeOut: TIME := TIME#500ms;
END_VAR

(*
MC_Power
Can Also be used MC_Reset, just trigger xEnable.
It is Highly Recommend to use OpenSML_Stop to force stop movements.
*)
Axis.ControlWord.2:=xEmergencyStop;//QuickStop
CASE iState OF
	0://start
		xDone:=FALSE;
		xError:=FALSE;
		Axis.ControlWord.0:=FALSE;//SwitchOn
		Axis.ControlWord.1:=FALSE;//EnableVoltage
		Axis.ControlWord.3:=FALSE;//EnableOperation
		Axis.ControlWord.7:=FALSE;//FaultReset
		IF xEnable THEN
			IF Axis.StatusWord.3 THEN iState:=10;//If there have error, Reset first
			ELSE iState:=20;//No error, go go
			END_IF
		END_IF
	10://reset
		Axis.ControlWord.7:=TRUE;//bit7 faultreset
		tonTimeout(IN:=TRUE,PT:=tTimeOut);
		IF tonTimeout.Q AND NOT Axis.StatusWord.3 THEN//not fault
			Axis.ControlWord.7:=FALSE;//bit7 faultreset
			tonTimeout(IN:=FALSE);
			iState:=20;
		ELSIF tonTimeout.Q THEN iState:=999;//error
		END_IF
	20://Enable Voltage
		Axis.ControlWord.1:=TRUE;
		tonTimeout(IN:=TRUE,PT:=tTimeOut);
		IF Axis.StatusWord.0 THEN//ReadyToSwitchOn
			tonTimeout(IN:=FALSE);
			iState:=30;
		ELSIF tonTimeout.Q THEN iState:=999;//error
		END_IF
	30://Switch ON
		Axis.ControlWord.0:=TRUE;
		tonTimeout(IN:=TRUE,pt:=tTimeOut);
		IF Axis.StatusWord.1 THEN
			tonTimeout(IN:=FALSE);
			iState:=40;
		ELSIF tonTimeout.Q THEN iState:=999;//error
		END_IF
	40://EnableOperation
		Axis.Target_Position:=Axis.Position_Actual_Value;
		Axis.ControlWord.3:=TRUE;
		tonTimeout(IN:=TRUE,pt:=tTimeOut);
		IF Axis.StatusWord.2 THEN
			tonTimeout(IN:=FALSE);
			iState:=50;
		ELSIF tonTimeout.Q THEN iState:=999;//error
		END_IF
	50://Success
		xDone:=TRUE;
		IF NOT xEnable THEN
			Axis.ControlWord.3:=FALSE;
			iState:=0;
		END_IF
		IF Axis.StatusWord.3 THEN
			iState:=999;//Error when running
		END_IF
	999://Error wait
		tonTimeout(IN:=FALSE);
		xError:=TRUE;
		IF NOT xEnable THEN
			iState:=0;
		END_IF
END_CASE

END_FUNCTION_BLOCK

// OpenSML_Stop
/// https://github.com/feecat/opensml 
FUNCTION_BLOCK OpenSML_Stop
VAR_IN_OUT
	Axis: OpenSML_Axis;
END_VAR
VAR_INPUT
	xStop: BOOL;
END_VAR

(*
MC_Stop
Software Stop, True=Stop
*)
Axis.ControlWord.8:=xStop;

END_FUNCTION_BLOCK

// OpenSML_Home
/// https://github.com/feecat/opensml 
FUNCTION_BLOCK OpenSML_Home
VAR_IN_OUT
	Axis: OpenSML_Axis;
END_VAR
VAR_INPUT
	xEnable: BOOL;
END_VAR
VAR_OUTPUT
	xDone: BOOL;
	xError: BOOL;
END_VAR
VAR
	iState: INT;
	tonTimeout: TON;
	Pos_Old: DINT;
END_VAR

(*
Home Function Block
Need Manually Write To SDO:
607C: Home Offset
6098: Home method
6099: Home Speeds*
609A: Home Acceleration

6099.01 - Home Speed for Search Limit Switch
6099.02 - Home Speed for Index Pulse
*)
CASE iState OF
	0:
		xDone:=FALSE;
		xError:=FALSE;
		IF xEnable AND Axis.StatusWord.1 AND Axis.StatusWord.2 AND Axis.Modes_of_operation_display = 6 AND NOT Axis.StatusWord.3 THEN//ready
			iState:=10;//go go
		ELSIF xEnable AND Axis.StatusWord.1 AND Axis.Modes_of_operation_display <> 6 THEN//need switch mode
			Axis.ControlWord.3:=FALSE;//drop down operation enabled
			iState:=10;
		ELSIF xEnable THEN
			iState:=999;//error
		END_IF
	10:
		Axis.ControlWord.4 := FALSE;//Reset reference bit
		Axis.Modes_of_operation:=6;//Home Mode
		Axis.ControlWord.3:=Axis.Modes_of_operation_display=6;//Success change mode, enable operation
		IF Axis.StatusWord.2 THEN//Operation Enabled
			iState:=20;
		END_IF
	20:
		Axis.ControlWord.4 := TRUE;//start reference
		tonTimeout(IN:=axis.Position_Actual_Value = Pos_Old, pt:=T#10S);//If Position didnt change, error
		Pos_Old:=Axis.Position_Actual_Value;
		IF Axis.StatusWord.12 THEN//If HomeAttained, Success
			tonTimeout(IN:=FALSE);
			Axis.ControlWord.4:=FALSE;
			Axis.Target_Position:=Axis.Position_Actual_Value;
			iState:=30;
		ELSIF tonTimeout.Q OR NOT xEnable OR Axis.StatusWord.3 OR Axis.StatusWord.13 THEN iState:=999;//error
		END_IF
	30:
		xDone:=TRUE;
		IF NOT xEnable THEN//Wait next home
			iState:=0;
		END_IF
	999:
		tonTimeout(IN:=FALSE);
		Axis.ControlWord.4:=FALSE;
		xError:=TRUE;
		IF NOT xEnable THEN
			iState:=0;
		END_IF
END_CASE

END_FUNCTION_BLOCK

// OpenSML_ProfilePosition
/// https://github.com/feecat/opensml 
FUNCTION_BLOCK OpenSML_ProfilePosition
VAR_IN_OUT
	Axis: OpenSML_Axis;
END_VAR
VAR_INPUT
	xEnable: BOOL;
	xExecute: BOOL;
	xContinueMove: BOOL;
	xRelativeMode: BOOL;
	diTargetPosition: DINT;
	udiProfileVelocity: UDINT;
END_VAR
VAR_OUTPUT
	xDone: BOOL;
	xBusy: BOOL;
	xMoving: BOOL;
	xError: BOOL;
END_VAR
VAR
	iState: INT;
	tonTimeout: TON;
	tTimeOut: TIME := TIME#200ms;
END_VAR

(*
Profile Position Mode (=1)
Manually Write To SDO or Write To PDO If Needed:
6083: Profile Acceleration
6084: Profile Deceleration
6085: Quick Stop Deceleration
*)
//Settings
Axis.ControlWord.5:=xContinueMove;//It means if 1st positon not arrived and there got 2st position, It Will No Deceleration And continues the movements.
Axis.ControlWord.6:=xRelativeMode;//0 is Absolute, 1 is Relative
Axis.ControlWord.4:=xExecute AND iState = 20;
xBusy:=iState=20 AND Axis.StatusWord.12 AND NOT Axis.StatusWord.10;//Acknowledge and not Reached
xDone:=iState=20 AND Axis.StatusWord.10 AND NOT Axis.StatusWord.13;//Target Reached and not Following Error
xMoving:=NOT Axis.StatusWord.14;//Not Standstill

CASE iState OF
	0://start
		xDone:=FALSE;
		xBusy:=FALSE;
		xError:=FALSE;
		IF xEnable AND Axis.StatusWord.1 AND Axis.StatusWord.2 AND Axis.Modes_of_operation_display = 1 AND NOT Axis.StatusWord.3 THEN//ready
			iState:=10;//go go
		ELSIF xEnable AND Axis.StatusWord.1 AND Axis.Modes_of_operation_display <> 1 THEN//need switch mode
			Axis.ControlWord.3:=FALSE;//drop down operation enabled
			iState:=10;
		ELSIF xEnable THEN
			iState:=999;//error
		END_IF
	10://Set Mode
		Axis.Modes_of_operation:=1;//Profile Position Mode
		Axis.ControlWord.3:=Axis.Modes_of_operation_display=1;//Success change mode, enable operation
		IF Axis.StatusWord.2 AND Axis.Modes_of_operation_display = 1 THEN//Operation Enabled, Mode Changed success
			iState:=20;
		END_IF
	20://Movement
		Axis.Profile_Velocity:=udiProfileVelocity;
		Axis.Target_Position:=diTargetPosition;
		IF Axis.StatusWord.13 OR Axis.StatusWord.3 THEN//Axis Error
			iState:=999;
		ELSIF NOT xEnable THEN
			Axis.Profile_Velocity:=0;
			Axis.Target_Position:=0;
			iState:=0;
		END_IF
	999://Error wait
		Axis.Profile_Velocity:=0;
		Axis.Target_Position:=0;
		tonTimeout(IN:=FALSE);
		xError:=TRUE;
		IF NOT xEnable THEN
			iState:=0;
		END_IF
END_CASE

END_FUNCTION_BLOCK

// OpenSML_ProfileVelocity
/// https://github.com/feecat/opensml 
FUNCTION_BLOCK OpenSML_ProfileVelocity
VAR_IN_OUT
	Axis: OpenSML_Axis;
END_VAR
VAR_INPUT
	xEnable: BOOL;
	diTargetVelocity: DINT;
END_VAR
VAR_OUTPUT
	xError: BOOL;
END_VAR
VAR
	iState: INT;
	tonTimeout: TON;
	tTimeOut: TIME := TIME#200ms;
END_VAR

(*
Profile Velocity Mode (=3)
Manually Write To SDO or Write To PDO If Needed:
6083: Profile Acceleration
6084: Profile Deceleration
6085: Quick Stop Deceleration
*)
CASE iState OF
	0://start
		xError:=FALSE;
		IF xEnable AND Axis.StatusWord.1 AND Axis.StatusWord.2 AND Axis.Modes_of_operation_display = 3 AND NOT Axis.StatusWord.3 THEN//ready
			iState:=10;//go go
		ELSIF xEnable AND Axis.StatusWord.1 AND Axis.Modes_of_operation_display <> 3 THEN//need switch mode
			Axis.ControlWord.3:=FALSE;//drop down operation enabled
			iState:=10;
		ELSIF xEnable THEN
			iState:=999;//error
		END_IF
	10://Set Mode
		Axis.Modes_of_operation:=3;//Profile Velocity Mode
		Axis.ControlWord.3:=Axis.Modes_of_operation_display=3;//Success change mode, enable operation
		IF Axis.StatusWord.2 AND Axis.Modes_of_operation_display = 3 THEN//Operation Enabled, Mode Changed success
			iState:=20;
		END_IF
	20://Movement
		Axis.Target_Velocity:=diTargetVelocity;
		IF Axis.StatusWord.3 THEN
			iState:=999;
		ELSIF NOT xEnable THEN
			Axis.Target_Velocity:=0;
			iState:=0;
		END_IF
	999://Error wait
		Axis.Target_Velocity:=0;
		tonTimeout(IN:=FALSE);
		xError:=TRUE;
		IF NOT xEnable THEN
			iState:=0;
		END_IF
END_CASE

END_FUNCTION_BLOCK

// OpenSML_SyncPosition
/// https://github.com/feecat/opensml 
FUNCTION_BLOCK OpenSML_SyncPosition
VAR_IN_OUT
	Axis: OpenSML_Axis;
END_VAR
VAR_INPUT
	MaxVelocity: LREAL := 2000;
	MaxAcceleration: LREAL := 200;
	MaxJerk: LREAL := 200;
	///0.001 = 1ms
	CycleTime: LREAL := 0.001;
	TargetPosition: LREAL;
	xEnable: BOOL;
	lrScale: LREAL := 1.0;
	xSimulation: BOOL;
END_VAR
VAR_OUTPUT
	xError: BOOL;
END_VAR
VAR
	otg: FB_S7RTT_OTG;
	iState: INT;
END_VAR

(*
Cyclic Synchronous Position Mode (=8)
Set 6060(Op mode) and 60C2(Interpolation time period) at Startup Parameters.

#####################################
NEED StruckigLight Library for Quadratic Velocity Ramp Calculate.

If in movement, Please DO NOT Drop down xEnable.
#####################################
*)

CASE iState OF
	0://start
		xError:=FALSE;
		IF xEnable AND Axis.StatusWord.1 AND Axis.StatusWord.2 AND Axis.Modes_of_operation_display = 8 AND NOT Axis.StatusWord.3 THEN//ready
			iState:=10;//go go
		ELSIF xEnable AND Axis.StatusWord.1 AND Axis.Modes_of_operation_display <> 8 THEN//need switch mode
			Axis.ControlWord.3:=FALSE;//drop down operation enabled, motor could free move
			iState:=10;
		ELSIF xSimulation THEN
			iState:=20;
		ELSIF xEnable THEN
			iState:=999;//error
		END_IF
	10://Set Mode
		Axis.Modes_of_operation:=8;//Cyclic Synchronous Position Mode
		Axis.ControlWord.3:=Axis.Modes_of_operation_display=8;//Success change mode, enable operation
		otg.CurrentPosition:=DINT_TO_LREAL(Axis.Position_Actual_Value) / lrScale;//Write actual position to otg
		IF Axis.StatusWord.2 AND Axis.Modes_of_operation_display = 8 THEN//Operation Enabled, Mode Changed success
			iState:=20;
		END_IF
	20://Movement
		otg(
			ControlInterface:= FALSE , 
			TargetPosition:= TargetPosition , 
			TargetVelocity:= 0 , 
			CycleTime:= CycleTime,
			MaxVelocity:= MaxVelocity , 
			MaxAcceleration:= MaxAcceleration , 
			MaxJerk:= MaxJerk);//accept new position and going on
			
		IF otg.NewPosition >= 0 THEN
			Axis.Target_Position := LREAL_TO_DINT(otg.NewPosition * lrScale);
		ELSE
			Axis.Target_Position := - LREAL_TO_DINT( - otg.NewPosition * lrScale);//it fix negative overflow problem.
		END_IF
		
		IF Axis.StatusWord.13 OR Axis.StatusWord.3 OR otg.xError THEN//Axis Error
			iState:=999;
		ELSIF NOT xEnable THEN
			iState:=0;
		END_IF
	999://Error wait
		xError:=TRUE;
		IF NOT xEnable THEN
			iState:=0;
		END_IF
END_CASE

END_FUNCTION_BLOCK

// OpenSML_SyncVelocity
/// https://github.com/feecat/opensml 
FUNCTION_BLOCK OpenSML_SyncVelocity
VAR_IN_OUT
	Axis: OpenSML_Axis;
END_VAR
VAR_INPUT
	MaxVelocity: LREAL := 2000;
	MaxAcceleration: LREAL := 200;
	MaxJerk: LREAL := 200;
	///0.001 = 1ms
	CycleTime: LREAL := 0.001;
	TargetVelocity: LREAL;
	xEnable: BOOL;
	lrScale: LREAL := 1.0;
	xSimulation: BOOL;
END_VAR
VAR_OUTPUT
	xError: BOOL;
END_VAR
VAR
	otg: FB_S7RTT_OTG;
	iState: INT;
END_VAR

(*
Normally we use CSP(=8) as CSV(=9) cus mostly servo dont have TargetVelocity PDO by default.
If you really want use CSV mode, Please connect OpenSML_SyncVelocity.otg.NewVelocity to TargetVelocity PDO after scale.

Cyclic Synchronous Position Mode (=8)
Set 6060(Op mode) and 60C2(Interpolation time period) at Startup Parameters.

#####################################
NEED StruckigLight Library for Quadratic Velocity Ramp Calculate.

If in movement, Please DO NOT Drop down xEnable.
#####################################
*)
CASE iState OF
	0://start
		xError:=FALSE;
		IF xEnable AND Axis.StatusWord.1 AND Axis.StatusWord.2 AND Axis.Modes_of_operation_display = 8 AND NOT Axis.StatusWord.3 THEN//ready
			iState:=10;//go go
		ELSIF xEnable AND Axis.StatusWord.1 AND Axis.Modes_of_operation_display <> 8 THEN//need switch mode
			Axis.ControlWord.3:=FALSE;//drop down operation enabled, motor could free move
			iState:=10;
		ELSIF xSimulation THEN
			iState:=20;
		ELSIF xEnable THEN
			iState:=999;//error
		END_IF
	10://Set Mode
		Axis.Modes_of_operation:=8;//Cyclic Synchronous Position Mode
		Axis.ControlWord.3:=Axis.Modes_of_operation_display=8;//Success change mode, enable operation
		otg.CurrentPosition:=DINT_TO_LREAL(Axis.Position_Actual_Value) / lrScale;//Write actual position to otg
		IF Axis.StatusWord.2 AND Axis.Modes_of_operation_display = 8 THEN//Operation Enabled, Mode Changed success
			iState:=20;
		END_IF
	20://Movement
		otg(
			ControlInterface:= TRUE , 
			TargetPosition:= 0 , 
			TargetVelocity:= TargetVelocity , 
			CycleTime:=CycleTime,
			MaxVelocity:= MaxVelocity , 
			MaxAcceleration:= MaxAcceleration , 
			MaxJerk:= MaxJerk);//accept new velocity and going on
			
		IF otg.NewPosition >= 0 THEN
			Axis.Target_Position := LREAL_TO_DINT(otg.NewPosition * lrScale);
		ELSE
			Axis.Target_Position := - LREAL_TO_DINT( - otg.NewPosition * lrScale);//it fix negative overflow problem.
		END_IF
		
		IF Axis.StatusWord.13 OR Axis.StatusWord.3 OR otg.xError THEN//Axis Error
			iState:=999;
		ELSIF NOT xEnable THEN
			iState:=0;
		END_IF
	999://Error wait
		xError:=TRUE;
		IF NOT xEnable THEN
			iState:=0;
		END_IF
END_CASE

END_FUNCTION_BLOCK

// OpenSML_TC3Link
/// https://github.com/feecat/opensml 
FUNCTION_BLOCK OpenSML_TC3Link
VAR_INPUT
	StatusWord AT %I*: UINT;
	Modes_of_operation_display AT %I*: SINT;
	Torque_Actual_Value AT %I*: INT;
	Position_Actual_Value AT %I*: DINT;
	Velocity_Actual_Value AT %I*: DINT;
	Current_Actual_Value AT %I*: INT;
	Following_Error_Actual_Value AT %I*: DINT;
END_VAR
VAR_OUTPUT
	ControlWord AT %Q*: UINT;
	Modes_of_operation AT %Q*: SINT;
	Target_Position AT %Q*: DINT;
	Profile_Velocity AT %Q*: UDINT;
	Target_Velocity AT %Q*: DINT;
	Target_torque AT %Q*: INT;
END_VAR
VAR_IN_OUT
	Axis: OpenSML_Axis;
END_VAR

(*******************************
For TwinCAT3, You can use TC3Link like below:

	VAR
		Axis_1: OpenSML_Axis;
		SyncPos: OpenSML_SyncPosition;
		link: OpenSML_TC3Link;
	END_VAR
	
	SyncPos(blablablabla);
	//Make sure link() call after other instance like OpenSML_SyncPosition.
	link(Axis:=Axis_1);

Then you can link variable to IO device like MAIN.link.Target_Position.
*******************************)
//Output							
	ControlWord        := Axis.ControlWord;
	Modes_of_operation := Axis.Modes_of_operation;
	Target_Position    := Axis.Target_Position;
	Profile_Velocity   := Axis.Profile_Velocity;
	Target_Velocity    := Axis.Target_Velocity;
	Target_torque      := Axis.Target_torque;
//Input							
	Axis.StatusWord                   := StatusWord;
	Axis.Modes_of_operation_display   := Modes_of_operation_display;
	Axis.Torque_Actual_Value          := Torque_Actual_Value;
	Axis.Position_Actual_Value        := Position_Actual_Value;
	Axis.Velocity_Actual_Value        := Velocity_Actual_Value;
	Axis.Current_Actual_Value         := Current_Actual_Value;
	Axis.Following_Error_Actual_Value := Following_Error_Actual_Value;

END_FUNCTION_BLOCK
